# EPICS autosave request: iocBoot/iocUSB1608G-2A0/auto_settings.req
file "1608G_settings.req", P=$(P)
